FUNCTION_BLOCK COMPLETE_LOOP
  (* Standard: 61499-2 *)
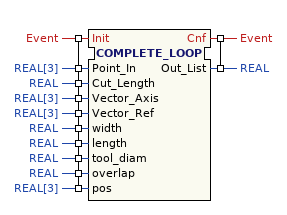
  EVENT_INPUT
    Init WITH Point_In, Cut_Length, Vector_Axis, Vector_Ref, width, length, tool_diam, overlap, pos;
  END_EVENT
  EVENT_OUTPUT
    Cnf WITH Out_List;
  END_EVENT
  VAR_INPUT
    Point_In : ARRAY [0..2] OF REAL;
    Cut_Length : REAL;
    Vector_Axis : ARRAY [0..2] OF REAL;
    Vector_Ref : ARRAY [0..2] OF REAL;
    width : REAL;
    length : REAL;
    tool_diam : REAL;
    overlap : REAL;
    pos : ARRAY [0..2] OF REAL;
  END_VAR
  VAR_OUTPUT
    Out_List : REAL;
  END_VAR
  FBS
    control_planes : CONTROL_PLANES;
    loop : LOOP_PLANAR_FACE;
    get_plane : GET_PLANE_EQUATION;
  END_FBS
  EVENT_CONNECTIONS
    Init TO control_planes.Init;
    loop.Cnf TO control_planes.Loop;
    get_plane.Cnf TO loop.Init;
    control_planes.Move TO get_plane.Init;
    control_planes.Finish TO Cnf;
  END_CONNECTIONS
  DATA_CONNECTIONS
    loop.Point_list TO Out_List;
    tool_diam TO loop.tool_diam;
    control_planes.Pos_Out TO loop.pos;
    overlap TO loop.overlap;
    length TO loop.length;
    get_plane.Plane TO loop.plane;
    width TO loop.width;
    Vector_Ref TO get_plane.Vector_Ref;
    Vector_Axis TO get_plane.Vector_Axis;
    control_planes.Point_Out TO get_plane.Point;
    Cut_Length TO control_planes.Cut_Length;
    Point_In TO control_planes.Point_In;
    Vector_Axis TO control_planes.Vector_Axis;
    pos TO control_planes.Pos_In;
  END_CONNECTIONS
END_FUNCTION_BLOCK
